FUNCTION_BLOCK FB_PointManager_PostgreSQL
VAR_OUTPUT
    bBusy : BOOL;
    bDone : BOOL;
    bError : BOOL;
    eResult : E_PointStoreResult := POINTSTORE_IDLE;
    nErrorID : UDINT;
    sLastOperation : STRING(80);
    bFound : BOOL;
    xPoint : ST_Point;
    pPoint : POINTER TO ST_Point;
END_VAR
VAR
    DB : FB_DBClient;
    nState : UINT := 0;

    sRobotPrefix : STRING(80);
    sPointDatabase : STRING(255);
    sSql : STRING(4095);

    sPendingName : STRING(80);
    sPendingNewName : STRING(80);
    sPendingNameExpression : STRING(255);
END_VAR

bDone := FALSE;
DB();

CASE nState OF
0:
    bBusy := FALSE;

10:
    bBusy := TRUE;
    eResult := POINTSTORE_BUSY;

    IF DB.ConfigurePostgreSQL(
        sDriver := DB.sDriver,
        sDatabaseServerNetID := DB.sDatabaseServerNetID,
        sServer := DB.sServer,
        nPort := DB.nPort,
        sDatabase := DB.sDatabase,
        sUser := DB.sUser,
        sPassword := DB.sPassword,
        sSchema := 'public'
    ) THEN
        ADSLOGSTR(ADSLOG_MSGTYPE_HINT, 'PointManager: database configuration accepted', '');
        nState := 20;
    END_IF

20:
    IF DB.bError THEN
        nErrorID := DB.nErrorID;
        sLastOperation := DB.sLastOperation;
        bError := TRUE;
        bBusy := FALSE;
        eResult := POINTSTORE_DATABASE_ERROR;
        nState := 0;
    ELSIF DB.bDone THEN
        nState := 30;
    END_IF

30:
    IF DB.Connect() THEN
        ADSLOGSTR(ADSLOG_MSGTYPE_HINT, 'PointManager: database connection accepted', '');
        nState := 40;
    END_IF

40:
    IF DB.bError THEN
        nErrorID := DB.nErrorID;
        sLastOperation := DB.sLastOperation;
        bError := TRUE;
        bBusy := FALSE;
        eResult := POINTSTORE_DATABASE_ERROR;
        nState := 0;
    ELSIF DB.bDone THEN
        bBusy := FALSE;
        eResult := POINTSTORE_DONE;
        bDone := TRUE;
        sLastOperation := 'Connected to point database';
        nState := 0;
    END_IF

100:
    IF DB.Execute(sSQL := sSql) THEN
        nState := 110;
    END_IF

110:
    IF DB.bError THEN
        nErrorID := DB.nErrorID;
        sLastOperation := DB.sLastOperation;
        bError := TRUE;
        bBusy := FALSE;
        eResult := POINTSTORE_DATABASE_ERROR;
        nState := 0;
    ELSIF DB.bDone THEN
        bBusy := FALSE;
        eResult := POINTSTORE_DONE;
        bDone := TRUE;
        sLastOperation := 'Point operation completed';
        nState := 0;
    END_IF

200:
    IF DB.Query(
        sSQL := sSql,
        pData := ADR(xPoint),
        cbData := SIZEOF(xPoint),
        nStartIndex := 0,
        nRecordCount := 1
    ) THEN
        nState := 210;
    END_IF

210:
    IF DB.bError THEN
        nErrorID := DB.nErrorID;
        sLastOperation := DB.sLastOperation;
        bError := TRUE;
        bBusy := FALSE;
        eResult := POINTSTORE_DATABASE_ERROR;
        nState := 0;
    ELSIF DB.bDone THEN
        bFound := xPoint.id <> 0;
        IF bFound THEN
            pPoint := ADR(xPoint);
        ELSE
            pPoint := 0;
        END_IF
        bBusy := FALSE;
        eResult := POINTSTORE_DONE;
        bDone := TRUE;
        sLastOperation := 'Point loaded';
        nState := 0;
    END_IF
END_CASE

METHOD PUBLIC Configure : BOOL
VAR_INPUT
    sPrefix : STRING(80);
    sDatabase : STRING(255);
END_VAR
Configure := FALSE;

IF (nState = 0) AND NOT bBusy AND (sPrefix <> '') AND (sDatabase <> '') THEN
    sRobotPrefix := sPrefix;
    sPointDatabase := sDatabase;
    bError := FALSE;
    nErrorID := 0;
    ADSLOGSTR(ADSLOG_MSGTYPE_HINT, 'PointManager.Configure accepted for %s', sPointDatabase);
    nState := 10;
    Configure := TRUE;
END_IF
END_METHOD

METHOD PUBLIC Create2D : BOOL
VAR_INPUT
    sName : STRING(80);
    pose : stPoseGeneral;
    frameId : UINT;
END_VAR
Create2D := FALSE;

IF (nState = 0) AND NOT bBusy AND DB.bConnected THEN
    IF sName = '' THEN
        sPendingNameExpression := SqlDefaultPointName();
    ELSE
        sPendingNameExpression := SqlQuotedLiteral(sName);
    END_IF

    sSql := 'INSERT INTO Point (robot_prefix, short_name, pose_kind, frame_id, x, y, z, rx, ry, rz, rz) VALUES (';
    sSql := CONCAT(sSql, SqlQuotedLiteral(sRobotPrefix));
    sSql := CONCAT(sSql, ', ');
    sSql := CONCAT(sSql, sPendingNameExpression);
    sSql := CONCAT(sSql, ', ');
    sSql := CONCAT(sSql, SqlQuotedLiteral('POSE_2D'));
    sSql := CONCAT(sSql, ', ');
    sSql := CONCAT(sSql, UINT_TO_STRING(frameId));
    sSql := CONCAT(sSql, ', ');
    sSql := CONCAT(sSql, LREAL_TO_STRING(pose.x));
    sSql := CONCAT(sSql, ', ');
    sSql := CONCAT(sSql, LREAL_TO_STRING(pose.y));
    sSql := CONCAT(sSql, ', NULL, NULL, NULL, NULL, ');
    sSql := CONCAT(sSql, LREAL_TO_STRING(pose.rz));
    sSql := CONCAT(sSql, ')');
    bError := FALSE;
    bBusy := TRUE;
    eResult := POINTSTORE_BUSY;
    sLastOperation := 'Create 2D point';
    nState := 100;
    Create2D := TRUE;
END_IF
END_METHOD

METHOD PUBLIC Create2DValues : BOOL
VAR_INPUT
        sName : STRING(80);
        x : LREAL;
        y : LREAL;
        rz : LREAL;
        frameId : UINT;
END_VAR
VAR
        pose : stPoseGeneral;
END_VAR
pose.x := x;
pose.y := y;
pose.rz := rz;

Create2DValues := Create2D(
        sName := sName,
        pose := pose,
        frameId := frameId
);
END_METHOD

METHOD PUBLIC Create3D : BOOL
VAR_INPUT
    sName : STRING(80);
    pose : stPoseGeneral;
    frameId : UINT;
END_VAR
Create3D := FALSE;

IF (nState = 0) AND NOT bBusy AND DB.bConnected THEN
    IF sName = '' THEN
        sPendingNameExpression := SqlDefaultPointName();
    ELSE
        sPendingNameExpression := SqlQuotedLiteral(sName);
    END_IF

    sSql := 'INSERT INTO Point (robot_prefix, short_name, pose_kind, frame_id, x, y, z, rx, ry, rz, rz) VALUES (';
    sSql := CONCAT(sSql, SqlQuotedLiteral(sRobotPrefix));
    sSql := CONCAT(sSql, ', ');
    sSql := CONCAT(sSql, sPendingNameExpression);
    sSql := CONCAT(sSql, ', ');
    sSql := CONCAT(sSql, SqlQuotedLiteral('POSE_3D'));
    sSql := CONCAT(sSql, ', ');
    sSql := CONCAT(sSql, UINT_TO_STRING(frameId));
    sSql := CONCAT(sSql, ', ');
    sSql := CONCAT(sSql, LREAL_TO_STRING(pose.x));
    sSql := CONCAT(sSql, ', ');
    sSql := CONCAT(sSql, LREAL_TO_STRING(pose.y));
    sSql := CONCAT(sSql, ', ');
    sSql := CONCAT(sSql, LREAL_TO_STRING(pose.z));
    sSql := CONCAT(sSql, ', ');
    sSql := CONCAT(sSql, LREAL_TO_STRING(pose.rx));
    sSql := CONCAT(sSql, ', ');
    sSql := CONCAT(sSql, LREAL_TO_STRING(pose.ry));
    sSql := CONCAT(sSql, ', ');
    sSql := CONCAT(sSql, LREAL_TO_STRING(pose.rz));
    sSql := CONCAT(sSql, ', NULL)');
    bError := FALSE;
    bBusy := TRUE;
    eResult := POINTSTORE_BUSY;
    sLastOperation := 'Create 3D point';
    nState := 100;
    Create3D := TRUE;
END_IF
END_METHOD

METHOD PUBLIC Create3DValues : BOOL
VAR_INPUT
        sName : STRING(80);
        x : LREAL;
        y : LREAL;
        z : LREAL;
        rx : LREAL;
        ry : LREAL;
        rz : LREAL;
        frameId : UINT;
END_VAR
VAR
        pose : stPoseGeneral;
END_VAR
pose.x := x;
pose.y := y;
pose.z := z;
pose.rx := rx;
pose.ry := ry;
pose.rz := rz;

Create3DValues := Create3D(
        sName := sName,
        pose := pose,
        frameId := frameId
);
END_METHOD

METHOD PUBLIC Delete : BOOL
VAR_INPUT
    sName : STRING(80);
END_VAR
Delete := FALSE;

IF (nState = 0) AND NOT bBusy AND DB.Connected AND (sName <> '') THEN
    sPendingName := sName;
    sSql := 'DELETE FROM Point WHERE robot_prefix = ';
    sSql := CONCAT(sSql, SqlQuotedLiteral(sRobotPrefix));
    sSql := CONCAT(sSql, ' AND short_name = ');
    sSql := CONCAT(sSql, SqlQuotedLiteral(sPendingName));
    bError := FALSE;
    bBusy := TRUE;
    eResult := POINTSTORE_BUSY;
    sLastOperation := 'Delete point';
    nState := 100;
    Delete := TRUE;
END_IF
END_METHOD

METHOD PUBLIC Load : BOOL
VAR_INPUT
    sName : STRING(80);
END_VAR
Load := FALSE;

IF (nState = 0) AND NOT bBusy AND DB.bConnected AND (sName <> '') THEN
    xPoint.id := 0;
    bFound := FALSE;
    pPoint := 0;
    sSql := 'SELECT id, robot_prefix, short_name, pose_kind, frame_id, x, y, COALESCE(z, 0), COALESCE(rx, 0), COALESCE(ry, 0), COALESCE(rz, 0), COALESCE(rz, 0) FROM Point WHERE robot_prefix = ';
    sSql := CONCAT(sSql, SqlQuotedLiteral(sRobotPrefix));
    sSql := CONCAT(sSql, ' AND short_name = ');
    sSql := CONCAT(sSql, SqlQuotedLiteral(sName));
    bError := FALSE;
    bBusy := TRUE;
    eResult := POINTSTORE_BUSY;
    sLastOperation := 'Load point';
    nState := 200;
    Load := TRUE;
END_IF
END_METHOD

METHOD PUBLIC Rename : BOOL
VAR_INPUT
    sOldName : STRING(80);
    sNewName : STRING(80);
END_VAR
Rename := FALSE;

IF (nState = 0) AND NOT bBusy AND DB.bConnected AND (sOldName <> '') AND (sNewName <> '') THEN
    sPendingName := sOldName;
    sPendingNewName := sNewName;
    sSql := 'UPDATE Point SET short_name = ';
    sSql := CONCAT(sSql, SqlQuotedLiteral(sPendingNewName));
    sSql := CONCAT(sSql, ' WHERE robot_prefix = ');
    sSql := CONCAT(sSql, SqlQuotedLiteral(sRobotPrefix));
    sSql := CONCAT(sSql, ' AND short_name = ');
    sSql := CONCAT(sSql, SqlQuotedLiteral(sPendingName));
    bError := FALSE;
    bBusy := TRUE;
    eResult := POINTSTORE_BUSY;
    sLastOperation := 'Rename point';
    nState := 100;
    Rename := TRUE;
END_IF
END_METHOD

METHOD PUBLIC Retouch2D : BOOL
VAR_INPUT
    sCurrentName : STRING(80);
    sNewName : STRING(80);
    pose : stPoseGeneral;
    frameId : UINT;
END_VAR
Retouch2D := FALSE;

IF (nState = 0) AND NOT bBusy AND DB.bConnected AND (sCurrentName <> '') THEN
    IF sNewName = '' THEN
        sPendingNewName := sCurrentName;
    ELSE
        sPendingNewName := sNewName;
    END_IF

    sSql := 'UPDATE Point SET short_name = ';
    sSql := CONCAT(sSql, SqlQuotedLiteral(sPendingNewName));
    sSql := CONCAT(sSql, ', pose_kind = ');
    sSql := CONCAT(sSql, SqlQuotedLiteral('POSE_2D'));
    sSql := CONCAT(sSql, ', frame_id = ');
    sSql := CONCAT(sSql, UINT_TO_STRING(frameId));
    sSql := CONCAT(sSql, ', x = ');
    sSql := CONCAT(sSql, LREAL_TO_STRING(pose.x));
    sSql := CONCAT(sSql, ', y = ');
    sSql := CONCAT(sSql, LREAL_TO_STRING(pose.y));
    sSql := CONCAT(sSql, ', z = NULL, rx = NULL, ry = NULL, rz = NULL, rz = ');
    sSql := CONCAT(sSql, LREAL_TO_STRING(pose.rz));
    sSql := CONCAT(sSql, ' WHERE robot_prefix = ');
    sSql := CONCAT(sSql, SqlQuotedLiteral(sRobotPrefix));
    sSql := CONCAT(sSql, ' AND short_name = ');
    sSql := CONCAT(sSql, SqlQuotedLiteral(sCurrentName));
    bError := FALSE;
    bBusy := TRUE;
    eResult := POINTSTORE_BUSY;
    sLastOperation := 'Retouch 2D point';
    nState := 100;
    Retouch2D := TRUE;
END_IF
END_METHOD

METHOD PUBLIC Retouch3D : BOOL
VAR_INPUT
    sCurrentName : STRING(80);
    sNewName : STRING(80);
    pose : stPoseGeneral;
    frameId : UINT;
END_VAR
Retouch3D := FALSE;

IF (nState = 0) AND NOT bBusy AND DB.bConnected AND (sCurrentName <> '') THEN
    IF sNewName = '' THEN
        sPendingNewName := sCurrentName;
    ELSE
        sPendingNewName := sNewName;
    END_IF

    sSql := 'UPDATE Point SET short_name = ';
    sSql := CONCAT(sSql, SqlQuotedLiteral(sPendingNewName));
    sSql := CONCAT(sSql, ', pose_kind = ');
    sSql := CONCAT(sSql, SqlQuotedLiteral('POSE_3D'));
    sSql := CONCAT(sSql, ', frame_id = ');
    sSql := CONCAT(sSql, UINT_TO_STRING(frameId));
    sSql := CONCAT(sSql, ', x = ');
    sSql := CONCAT(sSql, LREAL_TO_STRING(pose.x));
    sSql := CONCAT(sSql, ', y = ');
    sSql := CONCAT(sSql, LREAL_TO_STRING(pose.y));
    sSql := CONCAT(sSql, ', z = ');
    sSql := CONCAT(sSql, LREAL_TO_STRING(pose.z));
    sSql := CONCAT(sSql, ', rx = ');
    sSql := CONCAT(sSql, LREAL_TO_STRING(pose.rx));
    sSql := CONCAT(sSql, ', ry = ');
    sSql := CONCAT(sSql, LREAL_TO_STRING(pose.ry));
    sSql := CONCAT(sSql, ', rz = ');
    sSql := CONCAT(sSql, LREAL_TO_STRING(pose.rz));
    sSql := CONCAT(sSql, ', rz = NULL WHERE robot_prefix = ');
    sSql := CONCAT(sSql, SqlQuotedLiteral(sRobotPrefix));
    sSql := CONCAT(sSql, ' AND short_name = ');
    sSql := CONCAT(sSql, SqlQuotedLiteral(sCurrentName));
    bError := FALSE;
    bBusy := TRUE;
    eResult := POINTSTORE_BUSY;
    sLastOperation := 'Retouch 3D point';
    nState := 100;
    Retouch3D := TRUE;
END_IF
END_METHOD

METHOD PRIVATE SqlDefaultPointName : STRING(255)
SqlDefaultPointName := SqlQuotedLiteral('Point_');
SqlDefaultPointName := CONCAT(SqlDefaultPointName, ' || to_char(CURRENT_TIMESTAMP, ');
SqlDefaultPointName := CONCAT(SqlDefaultPointName, SqlQuotedLiteral('YYYYMMDD_HH24MISS'));
SqlDefaultPointName := CONCAT(SqlDefaultPointName, ')');
END_METHOD

METHOD PRIVATE SqlLiteral : STRING(255)
VAR_INPUT
    sValue : STRING(80);
END_VAR
VAR
    nIndex : UINT;
    sCharacter : STRING(1);
END_VAR
SqlLiteral := '';

FOR nIndex := 1 TO LEN(sValue) DO
    sCharacter := MID(sValue, 1, nIndex);
    IF sCharacter = '' THEN
        SqlLiteral := CONCAT(SqlLiteral, '');
    ELSE
        SqlLiteral := CONCAT(SqlLiteral, sCharacter);
    END_IF
END_FOR
END_METHOD

METHOD PRIVATE SqlQuotedLiteral : STRING(255)
VAR_INPUT
    sValue : STRING(80);
END_VAR
SqlQuotedLiteral := CONCAT('', SqlLiteral(sValue));
SqlQuotedLiteral := CONCAT(SqlQuotedLiteral, '');
END_METHOD

END_FUNCTION_BLOCK

(* stored: Version 1.1.0.1, ProductVersion 3.1.4026.18
   POU FB_PointManager_PostgreSQL: Id {b6db9b06-31bb-4ece-93a6-63e2ef2bfd14}, SpecialFunc None
   Method Configure: Id {9afd4f79-abdf-4d6f-9468-3b2de7adc2e6}
   Method Create2D: Id {4f3fb25a-3bd2-40cd-a02f-eafd7977a3bc}
   Method Create2DValues: Id {6d0a5501-4711-4b6e-a9cc-b700a08ef80d}
   Method Create3D: Id {1d1332d7-a54a-4f18-a922-ea688237a6ba}
   Method Create3DValues: Id {0876cf04-57a5-41cd-b61d-dd40d85d1c65}
   Method Delete: Id {32755b89-1880-44f7-b7ce-099449a3858d}
   Method Load: Id {7c6bd9ca-3847-4f94-a291-3f5a9b1e9f65}
   Method Rename: Id {dca2df38-9b43-4108-b7b3-e6dfb2a0b6ac}
   Method Retouch2D: Id {023b645f-9053-469d-b8aa-e7a57d6e3e16}
   Method Retouch3D: Id {1b756aff-0a9c-482d-bf16-03e8d39bfdc3}
   Method SqlDefaultPointName: Id {e98c178d-ae82-4782-babf-178872f406d1}
   Method SqlLiteral: Id {4c12c60f-e04a-42c8-befa-6531ad96cd6f}
   Method SqlQuotedLiteral: Id {d01b6355-a0cb-4988-a2f6-23b38844004f} *)
